FUNCTION_BLOCK MediaMovel
VAR_INPUT
	Input		:REAL;	//Valor de entrada para fazer a média
	Amostras	:INT;	//Quantidade de amostras do valor de entrada para fazer a média móvel
	Tempo		:DINT;	//Tempo de amostragem
END_VAR
VAR_OUTPUT
	Output	:REAL;	//Valor da média móvel
END_VAR
VAR
	ArrayValores	:ARRAY[0..100] OF REAL;
	iCounter: INT;
	Acumulador: REAL;
	TON_TempoAmostra: TON;
END_VAR

//Se a quantidade de amostras for menor que 1, esse valor é configurado
IF Amostras < 1 THEN
	Amostras := 1;
ELSIF Amostras > 100 THEN
	Amostras := 100;
END_IF

//Temporizador para amostragem
TON_TempoAmostra(IN:= NOT TON_TempoAmostra.Q, PT:= DINT_TO_TIME(Tempo * 1000), Q=> , ET=> );

IF TON_TempoAmostra.Q THEN
	FOR iCounter := 1 TO (Amostras - 1) BY 1 DO
		ArrayValores[iCounter] := ArrayValores[iCounter + 1];
	END_FOR
	ArrayValores[Amostras] := Input;
END_IF

//Acumula os valores do array
Acumulador := 0;
FOR iCounter := 1 TO Amostras BY 1 DO
	Acumulador := Acumulador + ArrayValores[iCounter];
END_FOR

//Calcula a saída
Output := Acumulador / Amostras;

END_FUNCTION_BLOCK

(* stored: Version 1.1.0.1, ProductVersion 3.1.4024.14
   POU MediaMovel: Id {e0e72de2-bf91-463f-a894-2302eb8bc077}, SpecialFunc None *)
